(* CODESYS project SingleElevator.project

Project tree, tasks and I/O mapping:
  Device : CODESYS Control Win V3, 3S - Smart Software Solutions GmbH, version 3.5.18.0
    application Application
      libraries: Standard, 3.5.18.0 (System)
      task MainTask (cyclic, interval t#20ms, priority 1) calls Simulation, GA_collector, PLC_PRG
      task VISU_TASK (cyclic, interval 100 ms, priority 31) calls VisuElems.Visu_Prg
      global variables GVL
      visualisation Visualization
      program Simulation [ST]
      function block Doors_GA [SFC]: _aReady_active, _aBusy_active, _aChiusura_active, _aApertura_active, _aApertura_exit, _aOpFinished_active, _aResetDone_active, _aChiusura_exit_1, _a_aInit_activeState
      program GA_collector [FBD]
      function block MovimentoVert_GA [SFC]: _aInit_active, _aReady_active, _aBusy_active, _aSalita_active, _aDiscesa_active, _aSalita_exit, _aDiscesa_exit
      program PLC_PRG [SFC]: _aOpenDoors1_active, _aInizio_homing_active, _aFinecorsa_active, _aRisalitaLenta_active, _aOpenDoors_active, _aHMI_wait_active, _aMoto_verticale_exit, _aOpenDoors_exit, _aOpenDoors1_exit, _aMemoria_chiamate_active, _aMoto_verticale_active_1, _aChiusura_P_exit, _aChiusura_P_active, _aMoto_verticale_entry
  text list GlobalTextList
*)

// Device/Application/GVL
//{attribute 'qualified_only'}
VAR_GLOBAL
(* Elevator managing variables*)
	Open: BOOL;				(* Sensor: the door is fully open*)
	Closed: BOOL;			(* Sensor: the door is fully closed*)
	LimitDown: BOOL;		(* Sensor: lower limit sensor, if TRUE the lift has reached the lower limit*)
	LimitUp: BOOL;			(* Sensor: upper limit sensor, if TRUE the lift has reached the upper limit*)
	DeckSensor: BOOL;		(* Sensor: if TRUE the cab is in proximity of a deck*)
	RampSensor: BOOL;		(* Sensor: if TRUE the cab is in proximity of a ramp*)
	Presence :BOOL; 		(* Sensor: if TRUE something blocks the door photocell*)
	Emergency: BOOL;		(* Input: if TRUE the emergency button has been pressed*)

	Closing: BOOL;			(* Actuator: if TRUE the door starts closing*)
	Opening: BOOL;			(* Actuator: the door starts opening*)
	Motor_on: BOOL;			(* Actuator: if TRUE the lift pulley motor start moving*)
	Up: BOOL;				(* Actuator parameter: if TRUE the lift moves upward, downward otherwise*)
	Vel: BOOL;				(* Actuator parameter: motor speed, if TRUE high speed, low speed otherwise*)


	Current: INT;  			(* Visualization: variable used to storage the current deck*)
    Destination: INT;		(* Visualization: variable used to storage the the destination deck*)
	EmergencyVis: BOOL; 	(* Visualization: if TRUE the emergency light is turned on*)

	InitialDeck: INT := 1;	(* Only for simulation: variable used to define the initial deck*)
	InitCycle: BOOL := FALSE;(* Only for simulation: used to execute the instruction at the first cycle*)
	Height: INT;			(* Only for simulation: elevator height*)
	DeckRest: INT;        	(* Only for simulation: division rest for generating deck sensor*)
	Memory: INT;
	RampRest: INT;			(* Only for simulation: division rest for generating the ramp position*)
	MemoryR: INT;
	Door: INT;				(* Only for simulation: to visualize the closing of the door*)
	Displacement: INT;		(* Only for simulation: lift displacement, dependent on the motor speed*)

 (*Inputs: internal panel variables*)
	PG: BOOL;
	P1: BOOL;
	P2: BOOL;
	P3: BOOL;
	P4: BOOL;
	P5: BOOL;
	P6: BOOL;
	P7: BOOL;

(*Visualization: internal panel variables used to turn on the LED*)
	PGVis: BOOL;
	P1Vis: BOOL;
	P2Vis: BOOL;
	P3Vis: BOOL;
	P4Vis: BOOL;
	P5Vis: BOOL;
	P6Vis: BOOL;
	P7Vis: BOOL;

(*Inputs: external panel variables*)
	UpDeckG: BOOL;
	UpDeck1: BOOL;
	UpDeck2: BOOL;
	UpDeck3: BOOL;
	UpDeck4: BOOL;
	UpDeck5: BOOL;
	UpDeck6: BOOL;
	DownDeck7: BOOL;
	DownDeck6: BOOL;
	DownDeck5: BOOL;
	DownDeck4: BOOL;
	DownDeck3: BOOL;
	DownDeck2: BOOL;
	DownDeck1: BOOL;

(*Visualization: external panel variables used to turn on the LED*)
	UpDeckGVis: BOOL;
	UpDeck1Vis: BOOL;
	UpDeck2Vis: BOOL;
	UpDeck3Vis: BOOL;
	UpDeck4Vis: BOOL;
	UpDeck5Vis: BOOL;
	UpDeck6Vis: BOOL;
	DownDeck7Vis: BOOL;
	DownDeck6Vis: BOOL;
	DownDeck5Vis: BOOL;
	DownDeck4Vis: BOOL;
	DownDeck3Vis: BOOL;
	DownDeck2Vis: BOOL;
	DownDeck1Vis: BOOL;

(*Only for simulation: variables used to simulate the fault on deck sensor*)
	SensorG: BOOL;				(* if TRUE the magnetic information for deck G is lost and the deck sensor cannot become TRUE*)
	Sensor1: BOOL;				(* if TRUE the magnetic information for deck 1 is lost and the deck sensor cannot become TRUE*)
	Sensor2: BOOL;
	Sensor3: BOOL;
	Sensor4: BOOL;
	Sensor5: BOOL;
	Sensor6: BOOL;
	Sensor7: BOOL;
	FaultSensorAlarm: BOOL; 	(* Visulaization: if TRUE alerts the user of a deck sensor fault*)

(*Only for simulation: variables used to simulate the fault on ramp sensor*)
	RampGUp: BOOL;
	Ramp1Down: BOOL;
	Ramp1Up:BOOL;
	Ramp2Down: BOOL;
	Ramp2Up:BOOL;
	Ramp3Down: BOOL;
	Ramp3Up:BOOL;
	Ramp4Down: BOOL;
	Ramp4Up:BOOL;
	Ramp5Down: BOOL;
	Ramp5Up:BOOL;
	Ramp6Down: BOOL;
	Ramp6Up:BOOL;
	Ramp7Down: BOOL;
	FaultRampAlarm: BOOL; 		(* Visulaization: if TRUE alerts the user of a ramp sensor fault*)
	SensorGOK: BOOL;
	Sensor1OK: BOOL;
	Sensor2OK: BOOL;
	Sensor6OK: BOOL;
	Sensor3OK: BOOL;
	Sensor4OK: BOOL;
	Sensor5OK: BOOL;
	Sensor7OK: BOOL;
	RampGUpOK: BOOL;
	Ramp1DownOK: BOOL;
	Ramp1UpOK: BOOL;
	Ramp2DownOK: BOOL;
	Ramp2UpOK: BOOL;
	Ramp3DownOK: BOOL;
	Ramp3UpOK: BOOL;
	Ramp4DownOK: BOOL;
	Ramp4UpOK: BOOL;
	Ramp5DownOK: BOOL;
	Ramp5UpOK: BOOL;
	Ramp6DownOK: BOOL;
	Ramp6UpOK: BOOL;
	Ramp7DownOK: BOOL;
	Ramp7UpOK: BOOL;
	Doors_GA_0: Doors_GA;
	MovimentoVert_GA_0: MovimentoVert_GA;
	Homing: BOOL;
END_VAR

// Device/Application/Simulation
PROGRAM Simulation
VAR
END_VAR

(* Initial position of the cab inside the hoistway. It is executed only at the first cycle.  *)
IF NOT GVL.InitCycle THEN
			GVL.InitCycle := TRUE ;
			GVL.Height := 20 * GVL.InitialDeck;
		    GVL.Door := 0;
			GVL.Current := GVL.Height / 20;
END_IF;

(* Elevator management, these instructions are executed each cycle time*)

(* Elevator door control. *)
IF GVL.Closing THEN
	GVL.Door := GVL.Door + 1;		(*Closing door management*)
	GVL.Open := FALSE;
END_IF

IF GVL.Door >= 60 THEN						(* Closed door limit*)
	GVL.Closed := TRUE;
END_IF

IF GVL.Opening THEN
	GVL.Door := GVL.Door - 1; 	(* Opening door management*)
	GVL.Closed := FALSE;
END_IF

IF GVL.Door <= 0 THEN							(* Open door limit*)
	GVL.Open := TRUE;
END_IF


(* Maximum and minimum management in the door simulation*)
IF GVL.Door < 0 THEN
	 GVL.Door := 0;
END_IF

IF GVL.Door > 60 THEN
	GVL.Door := 60;
END_IF


(* Control of the cab position inside the hostway. *)
(* Displacement definition for graphic visualization*)
IF GVL.Vel THEN 
	GVL.Displacement := 2;
ELSE 
	GVL.Displacement := 1;
END_IF


(* Height modification relying on direction and speed*)
IF GVL.Motor_on AND GVL.Up THEN
	GVL.Height := GVL.Height + GVL.Displacement;
	GVL.LimitDown := FALSE;
END_IF

IF GVL.Motor_on AND NOT GVL.Up THEN
	GVL.Height := GVL.Height - GVL.Displacement;
	GVL.LimitUp := FALSE;
END_IF


(* Limits for visualization*)
IF GVL.Height < -20 THEN
	GVL.Height := -20;
END_IF

IF GVL.Height > 160 THEN
	GVL.Height := 160;
END_IF

(* Limit sensors management*)
IF GVL.Height <= -10 THEN
	GVL.LimitDown := TRUE;
END_IF

IF GVL.Height >= 150 THEN
	 GVL.LimitUp := TRUE;
END_IF


(*-------------------------------------------------------------------*)
(*  Fault Management (Deck and Ramp Sensors)   *)
(*-------------------------------------------------------------------*)
(* Deck Sensor*)
(* Range of value where the deck sensor is active*)
IF ((GVL.Height >= -1) AND (GVL.Height <= 1)) THEN
	GVL.SensorGOK := TRUE;
ELSE  
	GVL.SensorGOK := FALSE;
END_IF

IF ((GVL.Height >= 20-1) AND (GVL.Height <= 20+1)) THEN
	GVL.Sensor1OK := TRUE;
ELSE  
	GVL.Sensor1OK := FALSE;
END_IF

IF ((GVL.Height >= 40-1) AND (GVL.Height <= 40+1)) THEN
	GVL.Sensor2OK := TRUE;
ELSE  
	GVL.Sensor2OK := FALSE;
END_IF

IF ((GVL.Height >= 60-1) AND (GVL.Height <= 60+1)) THEN
	GVL.Sensor3OK := TRUE;
ELSE  
	GVL.Sensor3OK := FALSE;
END_IF

IF ((GVL.Height >= 80-1) AND (GVL.Height <= 80+1)) THEN
	GVL.Sensor4OK := TRUE;
ELSE  
	GVL.Sensor4OK := FALSE;
END_IF

IF ((GVL.Height >= 100-1) AND (GVL.Height <= 100+1)) THEN
	GVL.Sensor5OK := TRUE;
ELSE   
	GVL.Sensor5OK := FALSE;
END_IF

IF ((GVL.Height >= 120-1) AND (GVL.Height <= 120+1)) THEN
	GVL.Sensor6OK := TRUE;
ELSE  
	GVL.Sensor6OK := FALSE;
END_IF

IF ((GVL.Height >= 140-1) AND (GVL.Height <= 140+1)) THEN
	GVL.Sensor7OK := TRUE;
ELSE  
	GVL.Sensor7OK := FALSE;
END_IF

GVL.DeckSensor := (GVL.SensorGOK AND NOT GVL.SensorG) OR
				    (GVL.Sensor1OK AND NOT GVL.Sensor1) OR
				    (GVL.Sensor2OK AND NOT GVL.Sensor2) OR
				    (GVL.Sensor3OK AND NOT GVL.Sensor3) OR
				    (GVL.Sensor4OK AND NOT GVL.Sensor4) OR
				    (GVL.Sensor5OK AND NOT GVL.Sensor5) OR
				    (GVL.Sensor6OK AND NOT GVL.Sensor6) OR
				    (GVL.Sensor7OK AND NOT GVL.Sensor7);

(* Ramp Sensor*)
(* Range of value where the ramp sensor is active*)
IF ((GVL.Height >= 5-1) AND (GVL.Height <= 5+1)) THEN
	GVL.RampGUpOK := TRUE;
ELSE 
	GVL.RampGUpOK := FALSE;
END_IF

(* Ramp close to deck 1*)
IF ((GVL.Height >= 15-1) AND (GVL.Height <= 15+1)) THEN
	GVL.Ramp1DownOK := TRUE;
ELSE 
	GVL.Ramp1DownOK := FALSE;
END_IF

IF ((GVL.Height >= 25-1) AND (GVL.Height <= 25+1)) THEN
	GVL.Ramp1UpOK := TRUE;
ELSE 
	GVL.Ramp1UpOK := FALSE;
END_IF

(* Ramp close to deck 2*)
IF ((GVL.Height >= 35-1) AND (GVL.Height <= 35+1)) THEN
	GVL.Ramp2DownOK := TRUE;
ELSE 
	GVL.Ramp2DownOK := FALSE;
END_IF

IF ((GVL.Height >= 45-1) AND (GVL.Height <= 45+1)) THEN
	GVL.Ramp2UpOK := TRUE;
ELSE 
	GVL.Ramp2UpOK := FALSE;
END_IF

(*Ramp close to deck  3*)
IF ((GVL.Height >= 55-1) AND (GVL.Height <= 55+1)) THEN
	GVL.Ramp3DownOK := TRUE;
ELSE 
	GVL.Ramp3DownOK := FALSE;
END_IF

IF ((GVL.Height >= 65-1) AND (GVL.Height <= 65+1)) THEN
	GVL.Ramp3UpOK := TRUE;
ELSE 
	GVL.Ramp3UpOK := FALSE;
END_IF

(* Ramp close to deck  4*)
IF ((GVL.Height >= 75-1) AND (GVL.Height <= 75+1)) THEN
	GVL.Ramp4DownOK := TRUE;
ELSE 
	GVL.Ramp4DownOK := FALSE;
END_IF

IF ((GVL.Height >= 85-1) AND (GVL.Height <= 85+1)) THEN
	GVL.Ramp4UpOK := TRUE;
ELSE 
	GVL.Ramp4UpOK:=FALSE;
END_IF

(* Ramp close to deck  5*)
IF ((GVL.Height >= 95-1) AND (GVL.Height <= 95+1)) THEN
	GVL.Ramp5DownOK := TRUE;
ELSE 
	GVL.Ramp5DownOK := FALSE;
END_IF

IF ((GVL.Height >= 105-1) AND (GVL.Height <= 105+1)) THEN
	GVL.Ramp5UpOK := TRUE;
ELSE
	GVL.Ramp5UpOK := FALSE;
END_IF

(* Ramp close to deck  6*)
IF ((GVL.Height >= 115-1) AND (GVL.Height <= 115+1)) THEN
	GVL.Ramp6DownOK := TRUE;
ELSE 
	GVL.Ramp6DownOK := FALSE;
END_IF

IF ((GVL.Height >= 125-1) AND (GVL.Height <= 125+1)) THEN
	GVL.Ramp6UpOK := TRUE;
ELSE 
	GVL.Ramp6UpOK := FALSE;
END_IF

(* Ramp close to deck  7*)
IF ((GVL.Height >= 135-1) AND (GVL.Height <= 135+1)) THEN
	GVL.Ramp7DownOK := TRUE;
ELSE 
	GVL.Ramp7DownOK := FALSE;
END_IF

GVL.RampSensor:=(GVL.RampGUpOK AND NOT GVL.RampGUp) OR 
								(GVL.Ramp1DownOK AND NOT GVL.Ramp1Down ) OR 
								(GVL.Ramp1UpOK AND NOT GVL.Ramp1Up ) OR
								(GVL.Ramp2DownOK AND NOT GVL.Ramp2Down ) OR 
								(GVL.Ramp2UpOK AND NOT GVL.Ramp2Up ) OR
								(GVL.Ramp3DownOK AND NOT GVL.Ramp3Down ) OR
 								(GVL.Ramp3UpOK AND NOT GVL.Ramp3Up ) OR
								(GVL.Ramp4DownOK AND NOT GVL.Ramp4Down ) OR
 								(GVL.Ramp4UpOK AND NOT GVL.Ramp4Up ) OR
								(GVL.Ramp5DownOK AND NOT GVL.Ramp5Down ) OR
 								(GVL.Ramp5UpOK AND NOT GVL.Ramp5Up ) OR
								(GVL.Ramp6DownOK AND NOT GVL.Ramp6Down ) OR
								(GVL.Ramp6UpOK AND NOT GVL.Ramp6Up ) OR
								(GVL.Ramp7DownOK AND NOT GVL.Ramp7Down );

END_PROGRAM

// Device/Application/GA_collector
PROGRAM GA_collector
VAR
END_VAR

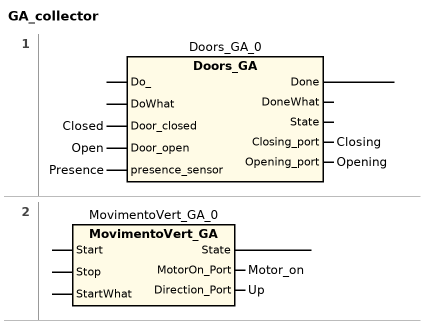
// NETWORK 1
Doors_GA_0(
    Door_closed := Closed,
    Door_open := Open,
    presence_sensor := Presence,
    Closing_port => Closing,
    Opening_port => Opening); // Doors_GA

// NETWORK 2
MovimentoVert_GA_0(MotorOn_Port => Motor_on, Direction_Port => Up); // MovimentoVert_GA

END_PROGRAM

// Device/Application/Doors_GA
FUNCTION_BLOCK Doors_GA
VAR_INPUT
	Do_: BOOL;
	DoWhat: STRING;
	Door_closed: BOOL;
	Door_open: BOOL;
	presence_sensor: BOOL;
END_VAR
VAR_OUTPUT
	Done: BOOL;
	DoneWhat: STRING;
    State: STRING;
	Closing_port: BOOL;
	Opening_port: BOOL;
END_VAR
VAR
END_VAR

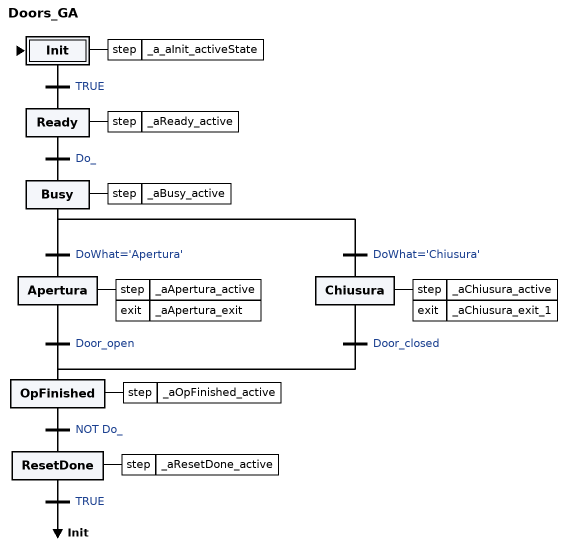
INITIAL_STEP Init:
    _a_aInit_activeState(N);  // step action
END_STEP
TRANSITION FROM Init TO Ready
    := TRUE;
END_TRANSITION
STEP Ready:
    _aReady_active(N);  // step action
END_STEP
TRANSITION FROM Ready TO Busy
    := Do_;
END_TRANSITION
STEP Busy:
    _aBusy_active(N);  // step action
END_STEP
TRANSITION FROM Busy TO Apertura
    := DoWhat='Apertura';
END_TRANSITION
STEP Apertura:
    _aApertura_active(N);  // step action
    _aApertura_exit(P0);  // exit action
END_STEP
TRANSITION FROM Apertura TO OpFinished
    := Door_open;
END_TRANSITION
TRANSITION FROM Busy TO Chiusura
    := DoWhat='Chiusura';
END_TRANSITION
STEP Chiusura:
    _aChiusura_active(N);  // step action
    _aChiusura_exit_1(P0);  // exit action
END_STEP
TRANSITION FROM Chiusura TO OpFinished
    := Door_closed;
END_TRANSITION
STEP OpFinished:
    _aOpFinished_active(N);  // step action
END_STEP
TRANSITION FROM OpFinished TO ResetDone
    := NOT Do_;
END_TRANSITION
STEP ResetDone:
    _aResetDone_active(N);  // step action
END_STEP
TRANSITION FROM ResetDone TO Init
    := TRUE;
END_TRANSITION

ACTION _aReady_active:
State := 'ready';
END_ACTION

ACTION _aBusy_active:
State := 'Busy';
END_ACTION

ACTION _aChiusura_active:
IF presence_sensor=FALSE AND Door_open=TRUE THEN
Closing_port:=TRUE;
Opening_port:=FALSE;
END_IF

IF presence_sensor= FALSE AND Door_closed=TRUE THEN
Closing_port:=FALSE;
END_IF

IF presence_sensor=TRUE THEN
	Closing_port:=FALSE;
	IF Door_open=FALSE THEN
    Opening_port:=TRUE;
	END_IF
	IF Door_open=TRUE THEN
	Opening_port:=FALSE;
	END_IF
END_IF
END_ACTION

ACTION _aApertura_active:
Opening_port :=TRUE;
END_ACTION

ACTION _aApertura_exit:
Opening_port := FALSE;
END_ACTION

ACTION _aOpFinished_active:
Done := TRUE;

IF door_open=TRUE THEN
	DoneWhat:='apertura';
END_IF

IF door_closed=TRUE THEN
	DoneWhat:='chiusura';
END_IF
END_ACTION

ACTION _aResetDone_active:
Done:=FALSE;
END_ACTION

ACTION _aChiusura_exit_1:
Closing_port := FALSE;
END_ACTION

ACTION _a_aInit_activeState:
State :='init';
END_ACTION

END_FUNCTION_BLOCK

// Device/Application/MovimentoVert_GA
FUNCTION_BLOCK MovimentoVert_GA
VAR_INPUT
	Start: BOOL;
	Stop: BOOL;
	StartWhat: STRING;
END_VAR
VAR_OUTPUT
	State: STRING;
	MotorOn_Port: BOOL;
	Direction_Port: BOOL;
END_VAR
VAR
END_VAR

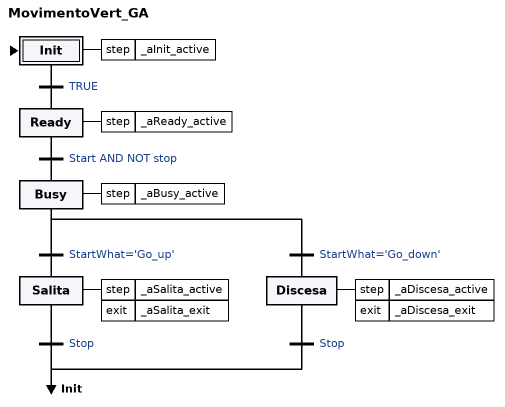
INITIAL_STEP Init:
    _aInit_active(N);  // step action
END_STEP
TRANSITION FROM Init TO Ready
    := TRUE;
END_TRANSITION
STEP Ready:
    _aReady_active(N);  // step action
END_STEP
TRANSITION FROM Ready TO Busy
    := Start AND NOT stop;
END_TRANSITION
STEP Busy:
    _aBusy_active(N);  // step action
END_STEP
TRANSITION FROM Busy TO Salita
    := StartWhat='Go_up';
END_TRANSITION
STEP Salita:
    _aSalita_active(N);  // step action
    _aSalita_exit(P0);  // exit action
END_STEP
TRANSITION FROM Salita TO Init
    := Stop;
END_TRANSITION
TRANSITION FROM Busy TO Discesa
    := StartWhat='Go_down';
END_TRANSITION
STEP Discesa:
    _aDiscesa_active(N);  // step action
    _aDiscesa_exit(P0);  // exit action
END_STEP
TRANSITION FROM Discesa TO Init
    := Stop;
END_TRANSITION

ACTION _aInit_active:
State:='init';
END_ACTION

ACTION _aReady_active:
State:='Ready';
END_ACTION

ACTION _aBusy_active:
State:='Busy';
END_ACTION

ACTION _aSalita_active:
Direction_Port := TRUE;
MotorOn_Port := TRUE;
END_ACTION

ACTION _aDiscesa_active:
Direction_Port := FALSE;
MotorOn_Port := TRUE;
END_ACTION

ACTION _aSalita_exit:
MotorOn_Port := FALSE;
END_ACTION

ACTION _aDiscesa_exit:
MotorOn_Port := FALSE;
END_ACTION

END_FUNCTION_BLOCK

// Device/Application/PLC_PRG
PROGRAM PLC_PRG
VAR
	OpComplete: BOOL;
	OpFinished: BOOL;
	OpDone: BOOL;
	OperationComplete: BOOL;
	Richiesta: BOOL;
	Coerent: INT;
	Libera: BOOL;
	OpFatta: BOOL;
	Current_Ok: BOOL;
	t_deck: INT := 0;
	Apertura_completata: BOOL;
	RR: INT;
	Check1: BOOL;
	RS_counter: INT := 0;
	Piano_partenza: INT;
	ok: BOOL;
	t_ramp: INT := 0;
	NuovaRichiesta: INT;
	Chiamata_in_sospeso: BOOL;
	VecchiaRichiesta: INT;
	Request_up: BOOL;
	Request_down: BOOL;
	Richiesta_interna: BOOL;
	RichiestaG: INT;
	Richiesta1: INT;
	Richiesta2: INT;
	Richiesta3: INT;
	Richiesta4: INT;
	Deck_counter: INT := 0;
	Ramp_counter: INT := 0;
	D_counter: INT := 0;
	t_finecorsa_alto: INT := 0;
	t_finecorsa_basso: INT := 0;
END_VAR

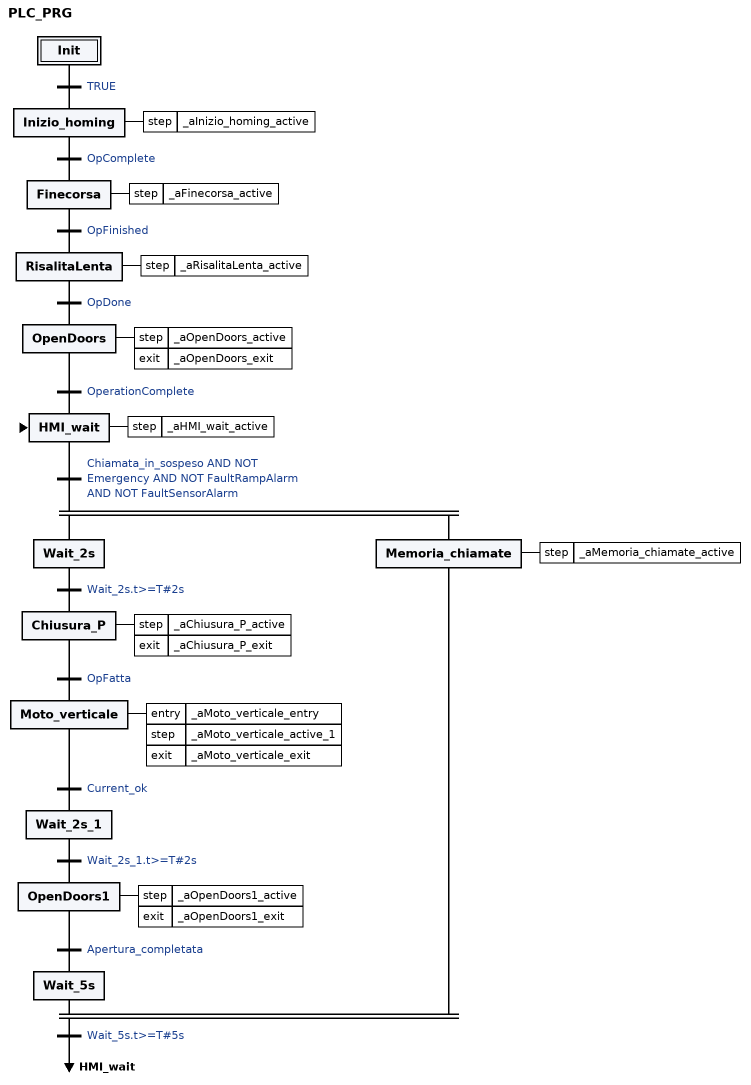
INITIAL_STEP Init:
END_STEP
TRANSITION FROM Init TO Inizio_homing
    := TRUE;
END_TRANSITION
STEP Inizio_homing:
    _aInizio_homing_active(N);  // step action
END_STEP
TRANSITION FROM Inizio_homing TO Finecorsa
    := OpComplete;
END_TRANSITION
STEP Finecorsa:
    _aFinecorsa_active(N);  // step action
END_STEP
TRANSITION FROM Finecorsa TO RisalitaLenta
    := OpFinished;
END_TRANSITION
STEP RisalitaLenta:
    _aRisalitaLenta_active(N);  // step action
END_STEP
TRANSITION FROM RisalitaLenta TO OpenDoors
    := OpDone;
END_TRANSITION
STEP OpenDoors:
    _aOpenDoors_active(N);  // step action
    _aOpenDoors_exit(P0);  // exit action
END_STEP
TRANSITION FROM OpenDoors TO HMI_wait
    := OperationComplete;
END_TRANSITION
STEP HMI_wait:
    _aHMI_wait_active(N);  // step action
END_STEP
TRANSITION FROM HMI_wait TO (Wait_2s, Memoria_chiamate)
    := Chiamata_in_sospeso AND NOT Emergency AND NOT FaultRampAlarm AND NOT FaultSensorAlarm;
END_TRANSITION
STEP Wait_2s:
END_STEP
TRANSITION FROM Wait_2s TO Chiusura_P
    := Wait_2s.t>=T#2s;
END_TRANSITION
STEP Chiusura_P:
    _aChiusura_P_active(N);  // step action
    _aChiusura_P_exit(P0);  // exit action
END_STEP
TRANSITION FROM Chiusura_P TO Moto_verticale
    := OpFatta;
END_TRANSITION
STEP Moto_verticale:
    _aMoto_verticale_entry(P1);  // entry action
    _aMoto_verticale_active_1(N);  // step action
    _aMoto_verticale_exit(P0);  // exit action
END_STEP
TRANSITION FROM Moto_verticale TO Wait_2s_1
    := Current_ok;
END_TRANSITION
STEP Wait_2s_1:
END_STEP
TRANSITION FROM Wait_2s_1 TO OpenDoors1
    := Wait_2s_1.t>=T#2s;
END_TRANSITION
STEP OpenDoors1:
    _aOpenDoors1_active(N);  // step action
    _aOpenDoors1_exit(P0);  // exit action
END_STEP
TRANSITION FROM OpenDoors1 TO Wait_5s
    := Apertura_completata;
END_TRANSITION
STEP Wait_5s:
END_STEP
STEP Memoria_chiamate:
    _aMemoria_chiamate_active(N);  // step action
END_STEP
TRANSITION FROM (Wait_5s, Memoria_chiamate) TO HMI_wait
    := Wait_5s.t>=T#5s;
END_TRANSITION

ACTION _aOpenDoors1_active:
IF Doors_GA_0.State='ready' THEN
	Doors_GA_0.Do_:=TRUE;
	Doors_GA_0.DoWhat:='Apertura';
END_IF

IF (Doors_GA_0.Done= TRUE) AND Doors_GA_0.State='Busy' THEN
	Doors_GA_0.Do_:=FALSE;
	Apertura_completata:=TRUE;
END_IF
END_ACTION

ACTION _aInizio_homing_active:
IF Doors_GA_0.State='ready' THEN
	Doors_GA_0.Do_:=TRUE;
	Doors_GA_0.DoWhat:='Chiusura';
END_IF

IF Doors_GA_0.Done= TRUE AND Doors_GA_0.State='Busy' THEN
	Doors_GA_0.Do_:=FALSE;
	OpComplete:=TRUE;
END_IF
END_ACTION

ACTION _aFinecorsa_active:
IF (LimitDown= FALSE) AND MovimentoVert_GA_0.State='Ready' THEN
    Vel:=FALSE;
	MovimentoVert_GA_0.Start:= TRUE;
	MovimentoVert_GA_0.StartWhat:='Go_down';
END_IF

IF LimitDown= TRUE THEN
	MovimentoVert_GA_0.Stop:= TRUE;
	OpFinished:= TRUE;
END_IF
END_ACTION

ACTION _aRisalitaLenta_active:
Vel:=FALSE;
IF MovimentoVert_GA_0.State='Ready'THEN
 IF DeckSensor= FALSE THEN
	MovimentoVert_GA_0.Stop:=FALSE;
	MovimentoVert_GA_0.Start:=TRUE;
	MovimentoVert_GA_0.StartWhat:='Go_up';
 END_IF
END_IF

IF DeckSensor= TRUE THEN
	MovimentoVert_GA_0.Stop:= TRUE;
	OpDone:=TRUE;
END_IF

//INIZIALIZZAZIONE
Current:=-1;
Chiamata_in_sospeso:=FALSE;
Current_Ok:=FALSE;
Richiesta:=FALSE;
END_ACTION

ACTION _aOpenDoors_active:
IF Doors_GA_0.State='ready' THEN
	Doors_GA_0.Do_:=TRUE;
	Doors_GA_0.DoWhat:='Apertura';
END_IF

IF (Doors_GA_0.Done= TRUE) AND Doors_GA_0.State='Busy' THEN
	Doors_GA_0.Do_:=FALSE;
	OperationComplete:=TRUE;
END_IF
END_ACTION

ACTION _aHMI_wait_active:
//EMERGENCY
IF Emergency =TRUE THEN
	EmergencyVis:=TRUE;
END_IF
IF Emergency = FALSE THEN
	EmergencyVis:=FALSE;
END_IF


//PULSANTIERA INTERNA

IF Chiamata_in_sospeso= FALSE THEN
	
IF PG= TRUE THEN
    Destination:=0; 
	PGVis:= TRUE;	
	Chiamata_in_sospeso:=TRUE;
END_IF

IF P1= TRUE THEN
    Destination:=1; 
	P1Vis:= TRUE;	
	Chiamata_in_sospeso:=TRUE;
END_IF

IF P2= TRUE THEN
    Destination:=2; 
	P2Vis:= TRUE;
	Chiamata_in_sospeso:=TRUE;
END_IF

IF P3= TRUE THEN
    Destination:=3; 
	P3Vis:= TRUE;	
	Chiamata_in_sospeso:=TRUE;
END_IF

IF P4= TRUE THEN
    Destination:=4; 
	P4Vis:= TRUE;	
	Chiamata_in_sospeso:=TRUE;
END_IF

IF P5= TRUE THEN
    Destination:=5; 
	P5Vis:= TRUE;	
	Chiamata_in_sospeso:=TRUE;
END_IF

IF P6= TRUE THEN
    Destination:=6; 
	P6Vis:= TRUE;	
	Chiamata_in_sospeso:=TRUE;
END_IF

IF P7=TRUE THEN
    Destination:=7; 
	P7Vis:= TRUE;	
	Chiamata_in_sospeso:=TRUE;
END_IF
END_IF
//Pulsantiera interna end

//Pulsantiera esterna, inizio up

IF UpDeckG=TRUE THEN
	UpDeckGVis:=TRUE;
    IF Chiamata_in_sospeso=FALSE THEN
	Destination:=0;
	Chiamata_in_sospeso:=TRUE;
	END_IF
END_IF

IF UpDeck1=TRUE THEN
	UpDeck1Vis:=TRUE;
    IF Chiamata_in_sospeso=FALSE THEN
	Destination:=1;
	Chiamata_in_sospeso:=TRUE;
	END_IF
END_IF

IF UpDeck2=TRUE THEN
	UpDeck2Vis:=TRUE;
    IF Chiamata_in_sospeso=FALSE THEN
	Destination:=2;
	Chiamata_in_sospeso:=TRUE;
	END_IF
END_IF

IF UpDeck3=TRUE THEN
	UpDeck3Vis:=TRUE;
    IF Chiamata_in_sospeso=FALSE THEN
	Destination:=3;
	Chiamata_in_sospeso:=TRUE;
	END_IF
END_IF

IF UpDeck4=TRUE THEN
	UpDeck4Vis:=TRUE;
    IF Chiamata_in_sospeso=FALSE THEN
	Destination:=4;
	Chiamata_in_sospeso:=TRUE;
	END_IF
END_IF

IF UpDeck5=TRUE THEN
	UpDeck5Vis:=TRUE;
    IF Chiamata_in_sospeso=FALSE THEN
	Destination:=5;
	Chiamata_in_sospeso:=TRUE;
	END_IF
END_IF

IF UpDeck6=TRUE THEN
	UpDeck6Vis:=TRUE;
    IF Chiamata_in_sospeso=FALSE THEN
	Destination:=6;
	Chiamata_in_sospeso:=TRUE;
	END_IF
END_IF

//Inizio down

IF DownDeck1=TRUE THEN
	DownDeck1Vis:=TRUE;
    IF Chiamata_in_sospeso=FALSE THEN
	Destination:=1;
	Chiamata_in_sospeso:=TRUE;
	END_IF
END_IF

IF DownDeck2=TRUE THEN
	DownDeck2Vis:=TRUE;
    IF Chiamata_in_sospeso=FALSE THEN
	Destination:=2;
	Chiamata_in_sospeso:=TRUE;
	END_IF
END_IF

IF DownDeck3=TRUE THEN
	DownDeck3Vis:=TRUE;
    IF Chiamata_in_sospeso=FALSE THEN
	Destination:=3;
	Chiamata_in_sospeso:=TRUE;
	END_IF
END_IF

IF DownDeck4=TRUE THEN
	DownDeck4Vis:=TRUE;
    IF Chiamata_in_sospeso=FALSE THEN
	Destination:=4;
	Chiamata_in_sospeso:=TRUE;
	END_IF
END_IF

IF DownDeck5=TRUE THEN
	DownDeck5Vis:=TRUE;
    IF Chiamata_in_sospeso=FALSE THEN
	Destination:=5;
	Chiamata_in_sospeso:=TRUE;
	END_IF
END_IF

IF DownDeck6=TRUE THEN
	DownDeck6Vis:=TRUE;
    IF Chiamata_in_sospeso=FALSE THEN
	Destination:=6;
	Chiamata_in_sospeso:=TRUE;
	END_IF
END_IF

IF DownDeck7=TRUE THEN
	DownDeck7Vis:=TRUE;
    IF Chiamata_in_sospeso=FALSE THEN
	Destination:=7;
	Chiamata_in_sospeso:=TRUE;
	END_IF
END_IF

//CHIAMATE IN SOSPESO TRAMITE VISUALIZER
IF  PGVis = TRUE
    OR	P1Vis = TRUE 
    OR	P2Vis = TRUE 
    OR	P3Vis = TRUE 
    OR  P4Vis = TRUE 
    OR  P5Vis = TRUE 
    OR	P6Vis = TRUE 
    OR	P7Vis = TRUE
	OR UpDeckGVis = TRUE
	OR UpDeck1Vis = TRUE
	OR UpDeck2Vis = TRUE
	OR UpDeck3Vis = TRUE
	OR UpDeck4Vis = TRUE
	OR UpDeck5Vis = TRUE
	OR UpDeck6Vis = TRUE
	OR DownDeck7Vis = TRUE
	OR DownDeck6Vis = TRUE
	OR DownDeck5Vis = TRUE
	OR DownDeck4Vis = TRUE
	OR DownDeck3Vis = TRUE
	OR DownDeck2Vis = TRUE
	OR DownDeck1Vis = TRUE THEN
	Chiamata_in_sospeso:=TRUE;
	ELSIF PGVis = FALSE
    OR	P1Vis = FALSE 
    OR	P2Vis = FALSE 
    OR	P3Vis = FALSE 
    OR  P4Vis = FALSE 
    OR  P5Vis = FALSE 
    OR	P6Vis = FALSE 
    OR	P7Vis = FALSE
	OR UpDeckGVis = FALSE
	OR UpDeck1Vis = FALSE
	OR UpDeck2Vis = FALSE
	OR UpDeck3Vis = FALSE
	OR UpDeck4Vis = FALSE
	OR UpDeck5Vis = FALSE
	OR UpDeck6Vis = FALSE
	OR DownDeck7Vis = FALSE
	OR DownDeck6Vis = FALSE
	OR DownDeck5Vis = FALSE
	OR DownDeck4Vis = FALSE
	OR DownDeck3Vis = FALSE
	OR DownDeck2Vis = FALSE
	OR DownDeck1Vis = FALSE THEN
	Chiamata_in_sospeso:=FALSE;
END_IF

(*IF Chiamata_in_sospeso=FALSE AND Current=-1 THEN
	Destination:=Current+1;
	ELSIF Current>-1 THEN Destination:=Current;
END_IF*)
END_ACTION

ACTION _aMoto_verticale_exit:
Richiesta:=FALSE;
END_ACTION

ACTION _aOpenDoors_exit:
OperationComplete:=FALSE;
Current_ok:= FALSE;
END_ACTION

ACTION _aOpenDoors1_exit:
Apertura_completata:=FALSE;
RS_counter:=0;

//Se abbiamo raggiunto il piano dobbiamo disattivare i led
IF P7Vis=TRUE AND Current=7 (*AND MovimentoVert_GA_0.State='Ready'*) THEN P7Vis:=FALSE;
ELSIF P6Vis=TRUE  AND Current=6 (*AND MovimentoVert_GA_0.State='Ready'*) THEN P6Vis:=FALSE;
ELSIF P5Vis=TRUE  AND Current=5 (*AND MovimentoVert_GA_0.State='Ready'*) THEN P5Vis:=FALSE;
ELSIF P4Vis=TRUE  AND Current=4 (*AND MovimentoVert_GA_0.State='Ready'*) THEN P4Vis:=FALSE;
ELSIF P3Vis=TRUE  AND Current=3 (*AND MovimentoVert_GA_0.State='Ready'*) THEN P3Vis:=FALSE;	
ELSIF P2Vis=TRUE  AND Current=2 (*AND MovimentoVert_GA_0.State='Ready'*) THEN P2Vis:=FALSE;
ELSIF P1Vis=TRUE  AND Current=1 (*AND MovimentoVert_GA_0.State='Ready'*) THEN P1Vis:=FALSE;	
ELSIF PGVis=TRUE  AND Current=0 (*AND MovimentoVert_GA_0.State='Ready'*) THEN PGVis:=FALSE;	
END_IF

IF UpDeck6Vis=TRUE AND Current=6 (*AND MovimentoVert_GA_0.State='Ready'*)  THEN UpDeck6Vis:=FALSE;
ELSIF UpDeck5Vis=TRUE  AND Current=5 (*AND MovimentoVert_GA_0.State='Ready'*)  THEN UpDeck5Vis:=FALSE;
ELSIF UpDeck4Vis=TRUE  AND Current=4 (*AND MovimentoVert_GA_0.State='Ready'*)  THEN UpDeck4Vis:=FALSE;
ELSIF UpDeck3Vis=TRUE  AND Current=3 (*AND MovimentoVert_GA_0.State='Ready'*)  THEN UpDeck3Vis:=FALSE;
ELSIF UpDeck2Vis=TRUE  AND Current=2 (*AND MovimentoVert_GA_0.State='Ready'*)  THEN UpDeck2Vis:=FALSE;
ELSIF UpDeck1Vis=TRUE  AND Current=1 (*AND MovimentoVert_GA_0.State='Ready'*)  THEN UpDeck1Vis:=FALSE;	
ELSIF UpDeckGVis=TRUE  AND Current=0 (*AND MovimentoVert_GA_0.State='Ready'*)  THEN UpDeckGVis:=FALSE;	
END_IF

IF DownDeck7Vis=TRUE  AND Current=7 (*AND MovimentoVert_GA_0.State='Ready'*)  THEN DownDeck7Vis:=FALSE;
ELSIF DownDeck6Vis=TRUE  AND Current=6 (*AND MovimentoVert_GA_0.State='Ready'*)  THEN DownDeck6Vis:=FALSE;
ELSIF DownDeck5Vis=TRUE  AND Current=5 (*AND MovimentoVert_GA_0.State='Ready'*)  THEN DownDeck5Vis:=FALSE;
ELSIF DownDeck4Vis=TRUE  AND Current=4 (*AND MovimentoVert_GA_0.State='Ready'*)  THEN DownDeck4Vis:=FALSE;
ELSIF DownDeck3Vis=TRUE  AND Current=3 (*AND MovimentoVert_GA_0.State='Ready'*)  THEN DownDeck3Vis:=FALSE;
ELSIF DownDeck2Vis=TRUE  AND Current=2 (*AND MovimentoVert_GA_0.State='Ready'*)  THEN DownDeck2Vis:=FALSE;
ELSIF DownDeck1Vis=TRUE  AND Current=1 (*AND MovimentoVert_GA_0.State='Ready'*)  THEN DownDeck1Vis:=FALSE;	
END_IF
END_ACTION

ACTION _aMemoria_chiamate_active:
//EMERGENCY AL VOLO
IF Emergency=TRUE THEN
	IF MovimentoVert_GA_0.StartWhat='Go_up' AND MovimentoVert_GA_0.State='Busy' AND RS_counter<2*(current-piano_partenza) THEN
		VEL:=FALSE;
		IF Current+1<Destination THEN
		Destination:=Current+1;
		END_IF
	END_IF
	
	IF MovimentoVert_GA_0.StartWhat='Go_down' AND MovimentoVert_GA_0.State='Busy' THEN
		VEL:=FALSE;
		IF Current-1>Destination THEN
		Destination:=Current-1;
		END_IF
	END_IF
	
END_IF

//FERMATA PER GUASTO DECK
IF DeckSensor=TRUE THEN
	Deck_counter:=0;
	Ramp_counter:=0;
END_IF

IF Ramp_counter=3 AND Deck_Counter=0 THEN
		VEL:=FALSE;
		FaultSensorAlarm:=TRUE;

	IF MovimentoVert_GA_0.StartWhat='Go_up' AND MovimentoVert_GA_0.State='Busy' THEN
		IF Current+1<Destination THEN
		Destination:=Current+1;
		END_IF
	END_IF
	
	IF MovimentoVert_GA_0.StartWhat='Go_down' AND MovimentoVert_GA_0.State='Busy' THEN
		IF Current-1>Destination THEN
		Destination:=Current-1;
		END_IF
	END_IF
	
END_IF


IF LimitUp=TRUE AND t_finecorsa_alto=0 THEN
	MovimentoVert_GA_0.Stop:=TRUE;
END_IF	

IF LimitUp=TRUE THEN t_finecorsa_alto:=t_finecorsa_alto+1; END_IF

IF LimitUp=TRUE AND t_finecorsa_alto=1 THEN
    Current:=8;
	Destination:=6;
	IF Current_ok=TRUE THEN
		FaultSensorAlarm:=TRUE;
	END_IF
END_IF

IF LimitDown=TRUE AND t_finecorsa_basso=0 THEN
	MovimentoVert_GA_0.Stop:=TRUE;
END_IF

IF LimitDown=TRUE THEN t_finecorsa_basso:=t_finecorsa_basso+1; END_IF

IF LimitDown=TRUE AND t_finecorsa_basso=1 THEN
	Current:=-1;
    Destination:=0;
	IF Current_ok=TRUE THEN
		FaultSensorAlarm:=TRUE;
	END_IF
END_IF

//FERMATA PER GUASTO RAMPA MOTO VERSO L'ALTO
IF RS_counter=1 AND Current=Piano_partenza+1 AND Destination<7 THEN
	VEL:=FALSE;
	FaultRampAlarm:=TRUE;
	Destination:=Current+1;
END_IF

IF RS_counter=3 AND Current=Piano_partenza+2 AND Destination<7 THEN
	VEL:=FALSE;
	FaultRampAlarm:=TRUE;
	Destination:=Current+1;
END_IF

IF RS_counter=5 AND Current=Piano_partenza+3 AND Destination<7 THEN
	VEL:=FALSE;
	FaultRampAlarm:=TRUE;
	Destination:=Current+1;
END_IF

IF RS_counter=7 AND Current=Piano_partenza+4 AND Destination<7 THEN
	VEL:=FALSE;
		FaultRampAlarm:=TRUE;
		Destination:=Current+1;
END_IF

IF RS_counter=9 AND Current=Piano_partenza+5 AND Destination<7 THEN
	VEL:=FALSE;
	FaultRampAlarm:=TRUE;
	IF DeckSensor=TRUE THEN	Destination:=Current+1; END_IF
END_IF

IF RS_counter=11 AND Current=Piano_partenza+6 AND Destination<7 THEN
	VEL:=FALSE;
		FaultRampAlarm:=TRUE;
		Destination:=Current+1;
END_IF

IF RS_counter=13 AND Current=Piano_partenza+7 THEN
	VEL:=FALSE;
	FaultRampAlarm:=TRUE;
END_IF

//FERMATA PER GUASTO RAMPA MOTO VERSO IL BASSO

IF RS_counter=1 AND Current=Piano_partenza-1 AND Destination>0 THEN
	VEL:=FALSE;
		FaultRampAlarm:=TRUE;
		Destination:=Current-1;
END_IF

IF RS_counter=3 AND Current=Piano_partenza-2 AND Destination>0 THEN
	VEL:=FALSE;
		FaultRampAlarm:=TRUE;
		Destination:=Current-1;
END_IF

IF RS_counter=5 AND Current=Piano_partenza-3 AND Destination>0 THEN
	VEL:=FALSE;
		FaultRampAlarm:=TRUE;
		Destination:=Current-1;
END_IF

IF RS_counter=7 AND Current=Piano_partenza-4 AND Destination>0 THEN
	VEL:=FALSE;
		FaultRampAlarm:=TRUE;
		Destination:=Current-1;
END_IF

IF RS_counter=9 AND Current=Piano_partenza-5 AND Destination>0 THEN
	VEL:=FALSE;
		FaultRampAlarm:=TRUE;
		Destination:=Current-1;
END_IF

IF RS_counter=11 AND Current=Piano_partenza-6 AND Destination>0 THEN
	VEL:=FALSE;
		FaultRampAlarm:=TRUE;
		Destination:=Current-1;
END_IF

IF RS_counter=13 AND Current=Piano_partenza-7 THEN
	VEL:=FALSE;
		FaultRampAlarm:=TRUE;
END_IF


//INIZIO PIANI AL VOLO
//Pulsantiera interna	
IF PG= TRUE THEN 
	PGVis:= TRUE;	
	Richiesta_interna:=TRUE;
END_IF

IF P1= TRUE THEN
	P1Vis:= TRUE;	
	Richiesta_interna:=TRUE;
END_IF

IF P2= TRUE THEN 
	P2Vis:= TRUE;
    Richiesta_interna:=TRUE;
END_IF

IF P3= TRUE THEN
	P3Vis:= TRUE;
    Richiesta_interna:=TRUE;
END_IF

IF P4= TRUE THEN
	P4Vis:= TRUE;	
	Richiesta_interna:=TRUE;
END_IF

IF P5= TRUE THEN
	P5Vis:= TRUE;	
	Richiesta_interna:=TRUE;
END_IF

IF P6= TRUE THEN 
	P6Vis:= TRUE;	
	Richiesta_interna:=TRUE;
END_IF

IF P7=TRUE THEN
	P7Vis:= TRUE;	
	Richiesta_interna:=TRUE;
END_IF


//Pulsantiera esterna, inizio up

IF UpDeckG=TRUE THEN
	UpDeckGVis:=TRUE;
    Request_up:=TRUE;
END_IF

IF UpDeck1=TRUE THEN
	UpDeck1Vis:=TRUE;
    Request_up:=TRUE;
END_IF

IF UpDeck2=TRUE THEN
	UpDeck2Vis:=TRUE;
    Request_up:=TRUE;
END_IF

IF UpDeck3=TRUE THEN
	UpDeck3Vis:=TRUE;
    Request_up:=TRUE;
END_IF

IF UpDeck4=TRUE THEN
	UpDeck4Vis:=TRUE;
    Request_up:=TRUE;
END_IF

IF UpDeck5=TRUE THEN
	UpDeck5Vis:=TRUE;
    Request_up:=TRUE;
END_IF

IF UpDeck6=TRUE THEN
	UpDeck6Vis:=TRUE;
    Request_up:=TRUE;
END_IF

//Inizio down

IF DownDeck1=TRUE THEN
	DownDeck1Vis:=TRUE;
    Request_down:=TRUE;
END_IF

IF DownDeck2=TRUE THEN
	DownDeck2Vis:=TRUE;
    Request_down:=TRUE;
END_IF

IF DownDeck3=TRUE THEN
	DownDeck3Vis:=TRUE;
    Request_down:=TRUE;
END_IF

IF DownDeck4=TRUE THEN
	DownDeck4Vis:=TRUE;
    Request_down:=TRUE;
END_IF

IF DownDeck5=TRUE THEN
	DownDeck5Vis:=TRUE;
    Request_down:=TRUE;
END_IF

IF DownDeck6=TRUE THEN
	DownDeck6Vis:=TRUE;
    Request_down:=TRUE;
END_IF

IF DownDeck7=TRUE THEN
	DownDeck7Vis:=TRUE;
    Request_down:=TRUE;
END_IF

//DEFINIZIONE REQUEST

IF DownDeck1Vis=FALSE AND DownDeck2Vis=FALSE AND DownDeck3Vis=FALSE AND DownDeck4Vis=FALSE AND DownDeck5Vis=FALSE AND DownDeck6Vis=FALSE AND DownDeck7Vis=FALSE THEN
    Request_Down:=FALSE;
END_IF 

IF UpDeckGVis=FALSE AND UpDeck1Vis=FALSE AND UpDeck2Vis=FALSE AND UpDeck3Vis=FALSE AND UpDeck4Vis=FALSE AND UpDeck5Vis=FALSE AND UpDeck6Vis=FALSE THEN
    Request_up:=FALSE;
END_IF 

IF PGvis=FALSE AND P1vis=FALSE AND P2vis=FALSE AND P3vis=FALSE AND P4vis=FALSE AND P5vis=FALSE AND P6vis=FALSE AND P7vis=FALSE THEN
    Richiesta_interna:=FALSE;
END_IF 


//CHIAMATE AL VOLO


//VIS INTERNI ALTO

IF MovimentoVert_GA_0.StartWhat='Go_up' AND MovimentoVert_GA_0.State='Busy' THEN
	IF Richiesta_interna=TRUE OR Request_up= TRUE THEN
	IF PGVis=TRUE THEN 
    IF 0<Destination AND Current<0 THEN
		Destination:=0;
		ELSIF 0>Destination AND Current_ok=TRUE THEN Destination:=0;
	END_IF
	END_IF
	END_IF
END_IF

IF MovimentoVert_GA_0.StartWhat='Go_up' AND MovimentoVert_GA_0.State='Busy' THEN
	IF Richiesta_interna=TRUE OR Request_up= TRUE THEN
	IF P1Vis=TRUE THEN 
    IF 1<Destination AND Current<1 THEN
		Destination:=1;
		ELSIF 1>Destination AND Current_ok=TRUE THEN Destination:=1;
	END_IF
	END_IF
	END_IF
END_IF

IF MovimentoVert_GA_0.StartWhat='Go_up' AND MovimentoVert_GA_0.State='Busy' THEN
	IF Richiesta_interna=TRUE OR Request_up= TRUE THEN
	IF P2Vis=TRUE THEN 
    IF 2<Destination AND Current<2 THEN
		Destination:=2;
		ELSIF 2>Destination AND Current_ok=TRUE THEN Destination:=2;
	END_IF
	END_IF
	END_IF
END_IF

IF MovimentoVert_GA_0.StartWhat='Go_up' AND MovimentoVert_GA_0.State='Busy' THEN
	IF Richiesta_interna=TRUE OR Request_up= TRUE THEN
	IF P3Vis=TRUE THEN 
    IF 3<Destination AND Current<3 THEN
		Destination:=3;
		ELSIF 3>Destination AND Current_ok=TRUE THEN Destination:=3;
	END_IF
	END_IF
	END_IF
END_IF

IF MovimentoVert_GA_0.StartWhat='Go_up' AND MovimentoVert_GA_0.State='Busy' THEN
	IF Richiesta_interna=TRUE OR Request_up= TRUE THEN
	IF P4Vis=TRUE THEN 
    IF 4<Destination AND Current<4 THEN
		Destination:=4;
		ELSIF 4>Destination AND Current_ok=TRUE THEN Destination:=4;
	END_IF
	END_IF
	END_IF
END_IF

IF MovimentoVert_GA_0.StartWhat='Go_up' AND MovimentoVert_GA_0.State='Busy' THEN
	IF Richiesta_interna=TRUE OR Request_up= TRUE THEN
	IF P5Vis=TRUE THEN 
    IF 5<Destination AND Current<5 THEN
		Destination:=5;
		ELSIF 5>Destination AND Current_ok=TRUE THEN Destination:=5;
	END_IF
	END_IF
	END_IF
END_IF

IF MovimentoVert_GA_0.StartWhat='Go_up' AND MovimentoVert_GA_0.State='Busy' THEN
	IF Richiesta_interna=TRUE OR Request_up= TRUE THEN
	IF P6Vis=TRUE THEN 
    IF 6<Destination AND Current<6 THEN
		Destination:=6;
		ELSIF 6>Destination AND Current_ok=TRUE THEN Destination:=6;
	END_IF
	END_IF
	END_IF
END_IF

IF MovimentoVert_GA_0.StartWhat='Go_up' AND MovimentoVert_GA_0.State='Busy' THEN
	IF Richiesta_interna=TRUE OR Request_up= TRUE THEN
	IF P7Vis=TRUE THEN 
    IF 7<Destination AND Current<7 THEN
		Destination:=7;
		ELSIF 7>Destination AND Current_ok=TRUE THEN Destination:=7;
	END_IF
	END_IF
	END_IF
END_IF


//VIS INTERNI DOWN
IF MovimentoVert_GA_0.StartWhat='Go_down' AND MovimentoVert_GA_0.State='Busy' THEN
	IF Richiesta_interna=TRUE OR Request_down= TRUE THEN
	IF PGVis=TRUE THEN 
    IF 0>Destination AND Current>0 THEN
		Destination:=0;
		ELSIF 0<Destination AND Current_ok=TRUE THEN Destination:=0;
	END_IF
	END_IF
	END_IF
END_IF

IF MovimentoVert_GA_0.StartWhat='Go_down' AND MovimentoVert_GA_0.State='Busy' THEN
	IF Richiesta_interna=TRUE OR Request_down= TRUE THEN
	IF P1Vis=TRUE THEN 
    IF 1>Destination AND Current>1 THEN
		Destination:=1;
		ELSIF 1<Destination AND Current_ok=TRUE THEN Destination:=1;
	END_IF
	END_IF
	END_IF
END_IF

IF MovimentoVert_GA_0.StartWhat='Go_down' AND MovimentoVert_GA_0.State='Busy' THEN
	IF Richiesta_interna=TRUE OR Request_down= TRUE THEN
	IF P2Vis=TRUE THEN 
    IF 2>Destination AND Current>2 THEN
		Destination:=2;
		ELSIF 2<Destination AND Current_ok=TRUE THEN Destination:=2;
	END_IF
	END_IF
	END_IF
END_IF

IF MovimentoVert_GA_0.StartWhat='Go_down' AND MovimentoVert_GA_0.State='Busy' THEN
	IF Richiesta_interna=TRUE OR Request_down= TRUE THEN
	IF P3Vis=TRUE THEN 
    IF 3>Destination AND Current>3 THEN
		Destination:=3;
		ELSIF 3<Destination AND Current_ok=TRUE THEN Destination:=3;
	END_IF
	END_IF
	END_IF
END_IF

IF MovimentoVert_GA_0.StartWhat='Go_down' AND MovimentoVert_GA_0.State='Busy' THEN
	IF Richiesta_interna=TRUE OR Request_down= TRUE THEN
	IF P4Vis=TRUE THEN 
    IF 4>Destination AND Current>4 THEN
		Destination:=4;
		ELSIF 4<Destination AND Current_ok=TRUE THEN Destination:=4;
	END_IF
	END_IF
	END_IF
END_IF

IF MovimentoVert_GA_0.StartWhat='Go_down' AND MovimentoVert_GA_0.State='Busy' THEN
	IF Richiesta_interna=TRUE OR Request_down= TRUE THEN
	IF P5Vis=TRUE THEN 
    IF 5>Destination AND Current>5 THEN
		Destination:=5;
		ELSIF 5<Destination AND Current_ok=TRUE THEN Destination:=5;
	END_IF
	END_IF
	END_IF
END_IF

IF MovimentoVert_GA_0.StartWhat='Go_down' AND MovimentoVert_GA_0.State='Busy' THEN
	IF Richiesta_interna=TRUE OR Request_down= TRUE THEN
	IF P6Vis=TRUE THEN 
    IF 6>Destination AND Current>6 THEN
		Destination:=6;
		ELSIF 6<Destination AND Current_ok=TRUE THEN Destination:=6;
	END_IF
	END_IF
	END_IF
END_IF

IF MovimentoVert_GA_0.StartWhat='Go_down' AND MovimentoVert_GA_0.State='Busy' THEN
	IF Richiesta_interna=TRUE OR Request_down= TRUE THEN
	IF P7Vis=TRUE THEN 
    IF 7>Destination AND Current>7 THEN
		Destination:=7;
		ELSIF 7<Destination AND Current_ok=TRUE THEN Destination:=7;
	END_IF
	END_IF
	END_IF
END_IF







//VIS ESTERNI UP

IF MovimentoVert_GA_0.StartWhat='Go_up' AND MovimentoVert_GA_0.State='Busy' THEN
	IF Richiesta_interna=TRUE OR Request_up= TRUE THEN
	IF UpDeckGVis=TRUE THEN 
    IF 0<Destination AND Current<0 THEN
		Destination:=0;
		ELSIF 0>Destination AND Current_ok=TRUE THEN Destination:=0;
	END_IF
	END_IF
	END_IF
END_IF

IF MovimentoVert_GA_0.StartWhat='Go_up' AND MovimentoVert_GA_0.State='Busy' THEN
	IF Richiesta_interna=TRUE OR Request_up= TRUE THEN
	IF UpDeck1Vis=TRUE THEN 
    IF 1<Destination AND Current<1 AND RS_counter<(2*(1-Piano_partenza)) THEN
		Destination:=1;
		ELSIF 1>Destination AND Current_ok=TRUE THEN Destination:=1;
	END_IF
	END_IF
	END_IF
END_IF

IF MovimentoVert_GA_0.StartWhat='Go_up' AND MovimentoVert_GA_0.State='Busy' THEN
	IF Richiesta_interna=TRUE OR Request_up= TRUE THEN
	IF UpDeck2Vis=TRUE THEN 
    IF 2<Destination AND Current<2 AND RS_counter<(2*(2-Piano_partenza)) THEN
		Destination:=2;
		ELSIF 2>Destination AND Current_ok=TRUE THEN Destination:=2;
	END_IF
	END_IF
	END_IF
END_IF

IF MovimentoVert_GA_0.StartWhat='Go_up' AND MovimentoVert_GA_0.State='Busy' THEN
	IF Richiesta_interna=TRUE OR Request_up= TRUE THEN
	IF UpDeck3Vis=TRUE THEN 
    IF 3<Destination AND Current<3 AND RS_counter<(2*(3-Piano_partenza)) THEN
		Destination:=3;
		ELSIF 3>Destination AND Current_ok=TRUE THEN Destination:=3;
	END_IF
	END_IF
	END_IF
END_IF

IF MovimentoVert_GA_0.StartWhat='Go_up' AND MovimentoVert_GA_0.State='Busy' THEN
	IF Richiesta_interna=TRUE OR Request_up= TRUE THEN
	IF UpDeck4Vis=TRUE THEN 
    IF 4<Destination AND Current<4 AND RS_counter<(2*(4-Piano_partenza)) THEN
		Destination:=4;
		ELSIF 4>Destination AND Current_ok=TRUE THEN Destination:=4;
	END_IF
	END_IF
	END_IF
END_IF

IF MovimentoVert_GA_0.StartWhat='Go_up' AND MovimentoVert_GA_0.State='Busy' THEN
	IF Richiesta_interna=TRUE OR Request_up= TRUE THEN
	IF UpDeck5Vis=TRUE THEN 
    IF 5<Destination AND Current<5 AND RS_counter<(2*(5-Piano_partenza)) THEN
		Destination:=5;
		ELSIF 5>Destination AND Current_ok=TRUE THEN Destination:=5;
	END_IF
	END_IF
	END_IF
END_IF

IF MovimentoVert_GA_0.StartWhat='Go_up' AND MovimentoVert_GA_0.State='Busy' THEN
	IF Richiesta_interna=TRUE OR Request_up= TRUE THEN
	IF UpDeck6Vis=TRUE THEN 
    IF 6<Destination AND Current<6 AND RS_counter<(2*(6-Piano_partenza)) THEN
		Destination:=6;
		ELSIF 6>Destination AND Current_ok=TRUE THEN Destination:=6;
	END_IF
	END_IF
	END_IF
END_IF

//VIS ESTERNI DOWN

IF MovimentoVert_GA_0.StartWhat='Go_down' AND MovimentoVert_GA_0.State='Busy' THEN
	IF Richiesta_interna=TRUE OR Request_down= TRUE THEN
	IF DownDeck1Vis=TRUE THEN 
    IF 1>Destination AND Current>1 AND RS_counter<(2*(Piano_partenza-1)) THEN
		Destination:=1;
		ELSIF 1<Destination AND Current_ok=TRUE THEN Destination:=1;
	END_IF
	END_IF
	END_IF
END_IF

IF MovimentoVert_GA_0.StartWhat='Go_down' AND MovimentoVert_GA_0.State='Busy' THEN
	IF Richiesta_interna=TRUE OR Request_down= TRUE THEN
	IF DownDeck2Vis=TRUE THEN 
    IF 2>Destination AND Current>2 AND RS_counter<(2*(Piano_partenza-2)) THEN
		Destination:=2;
		ELSIF 2<Destination AND Current_ok=TRUE THEN Destination:=2;
	END_IF
	END_IF
	END_IF
END_IF

IF MovimentoVert_GA_0.StartWhat='Go_down' AND MovimentoVert_GA_0.State='Busy' THEN
	IF Richiesta_interna=TRUE OR Request_down= TRUE THEN
	IF DownDeck3Vis=TRUE THEN 
    IF 3>Destination AND Current>3 AND RS_counter<(2*(Piano_partenza-3)) THEN
		Destination:=3;
		ELSIF 3<Destination AND Current_ok=TRUE THEN Destination:=3;
	END_IF
	END_IF
	END_IF
END_IF

IF MovimentoVert_GA_0.StartWhat='Go_down' AND MovimentoVert_GA_0.State='Busy' THEN
	IF Richiesta_interna=TRUE OR Request_down= TRUE THEN
	IF DownDeck4Vis=TRUE THEN 
    IF 4>Destination AND Current>4 AND RS_counter<(2*(Piano_partenza-4)) THEN
		Destination:=4;
		ELSIF 4<Destination AND Current_ok=TRUE THEN Destination:=4;
	END_IF
	END_IF
	END_IF
END_IF

IF MovimentoVert_GA_0.StartWhat='Go_down' AND MovimentoVert_GA_0.State='Busy' THEN
	IF Richiesta_interna=TRUE OR Request_down= TRUE THEN
	IF DownDeck5Vis=TRUE THEN 
    IF 5>Destination AND Current>5 AND RS_counter<(2*(Piano_partenza-5)) THEN
		Destination:=5;
		ELSIF 5<Destination AND Current_ok=TRUE THEN Destination:=5;
	END_IF
	END_IF
	END_IF
END_IF

IF MovimentoVert_GA_0.StartWhat='Go_down' AND MovimentoVert_GA_0.State='Busy' THEN
	IF Richiesta_interna=TRUE OR Request_down= TRUE THEN
	IF DownDeck6Vis=TRUE THEN 
    IF 6>Destination AND Current>6 AND RS_counter<(2*(Piano_partenza-6)) THEN
		Destination:=6;
		ELSIF 6<Destination AND Current_ok=TRUE THEN Destination:=6;
	END_IF
	END_IF
	END_IF
END_IF

IF MovimentoVert_GA_0.StartWhat='Go_down' AND MovimentoVert_GA_0.State='Busy' THEN
	IF Richiesta_interna=TRUE OR Request_down= TRUE THEN
	IF DownDeck7Vis=TRUE THEN 
    IF 7>Destination AND Current>7 THEN
		Destination:=7;
		ELSIF 7<Destination AND Current_ok=TRUE THEN Destination:=7;
	END_IF
	END_IF
	END_IF
END_IF


//MEMORIA CHIAMATE NON AL VOLO ESTERNO ALTO

IF MovimentoVert_GA_0.State='Ready' AND Chiamata_in_sospeso=TRUE THEN
	IF Richiesta_interna=TRUE OR Request_up= TRUE THEN
	IF UpDeckGVis=TRUE THEN 
    IF 0<Destination AND Current<0 THEN
		Destination:=0;
		ELSIF 0>Destination AND Current_ok=TRUE THEN Destination:=0;
	END_IF
	END_IF
	END_IF
END_IF

IF MovimentoVert_GA_0.State='Ready' AND Chiamata_in_sospeso=TRUE THEN
	IF Richiesta_interna=TRUE OR Request_up= TRUE THEN
	IF UpDeck1Vis=TRUE THEN 
    IF 1<Destination AND Current<1 THEN
		Destination:=1;
		ELSIF 1>Destination AND Current_ok=TRUE THEN Destination:=1;
	END_IF
	END_IF
	END_IF
END_IF

IF MovimentoVert_GA_0.State='Ready' AND Chiamata_in_sospeso=TRUE THEN
	IF Richiesta_interna=TRUE OR Request_up= TRUE THEN
	IF UpDeck2Vis=TRUE THEN 
    IF 2<Destination AND Current<2 THEN
		Destination:=2;
		ELSIF 2>Destination AND Current_ok=TRUE THEN Destination:=2;
	END_IF
	END_IF
	END_IF
END_IF

IF MovimentoVert_GA_0.State='Ready' AND Chiamata_in_sospeso=TRUE THEN
	IF Richiesta_interna=TRUE OR Request_up= TRUE THEN
	IF UpDeck3Vis=TRUE THEN 
    IF 3<Destination AND Current<3 THEN
		Destination:=3;
		ELSIF 3>Destination AND Current_ok=TRUE THEN Destination:=3;
	END_IF
	END_IF
	END_IF
END_IF

IF MovimentoVert_GA_0.State='Ready' AND Chiamata_in_sospeso=TRUE THEN
	IF Richiesta_interna=TRUE OR Request_up= TRUE THEN
	IF UpDeck4Vis=TRUE THEN 
    IF 4<Destination AND Current<4 THEN
		Destination:=4;
		ELSIF 4>Destination AND Current_ok=TRUE THEN Destination:=4;
	END_IF
	END_IF
	END_IF
END_IF

IF MovimentoVert_GA_0.State='Ready' AND Chiamata_in_sospeso=TRUE THEN
	IF Richiesta_interna=TRUE OR Request_up= TRUE THEN
	IF UpDeck5Vis=TRUE THEN 
    IF 5<Destination AND Current<5 THEN
		Destination:=5;
		ELSIF 5>Destination AND Current_ok=TRUE THEN Destination:=5;
	END_IF
	END_IF
	END_IF
END_IF

IF MovimentoVert_GA_0.State='Ready' AND Chiamata_in_sospeso=TRUE THEN
	IF Richiesta_interna=TRUE OR Request_up= TRUE THEN
	IF UpDeck6Vis=TRUE THEN 
    IF 6<Destination AND Current<6 THEN
		Destination:=6;
		ELSIF 6>Destination AND Current_ok=TRUE THEN Destination:=6;
	END_IF
	END_IF
	END_IF
END_IF

//MEMORIA CHIAMATE ESTERNO BASSO

IF MovimentoVert_GA_0.State='Ready' AND Chiamata_in_sospeso=TRUE THEN
	IF Richiesta_interna=TRUE OR Request_down= TRUE THEN
	IF DownDeck1Vis=TRUE THEN 
    IF 1>Destination AND Current>1 THEN
		Destination:=1;
		ELSIF 1<Destination AND Current_ok=TRUE THEN Destination:=1;
	END_IF
	END_IF
	END_IF
END_IF

IF MovimentoVert_GA_0.State='Ready' AND Chiamata_in_sospeso=TRUE THEN
	IF Richiesta_interna=TRUE OR Request_down= TRUE THEN
	IF DownDeck2Vis=TRUE THEN 
    IF 2>Destination AND Current>2 THEN
		Destination:=2;
		ELSIF 2<Destination AND Current_ok=TRUE THEN Destination:=2;
	END_IF
	END_IF
	END_IF
END_IF

IF MovimentoVert_GA_0.State='Ready' AND Chiamata_in_sospeso=TRUE THEN
	IF Richiesta_interna=TRUE OR Request_down= TRUE THEN
	IF DownDeck3Vis=TRUE THEN 
    IF 3>Destination AND Current>3 THEN
		Destination:=3;
		ELSIF 3<Destination AND Current_ok=TRUE THEN Destination:=3;
	END_IF
	END_IF
	END_IF
END_IF

IF MovimentoVert_GA_0.State='Ready' AND Chiamata_in_sospeso=TRUE THEN
	IF Richiesta_interna=TRUE OR Request_down= TRUE THEN
	IF DownDeck4Vis=TRUE THEN 
    IF 4>Destination AND Current>4 THEN
		Destination:=4;
		ELSIF 4<Destination AND Current_ok=TRUE THEN Destination:=4;
	END_IF
	END_IF
	END_IF
END_IF

IF MovimentoVert_GA_0.State='Ready' AND Chiamata_in_sospeso=TRUE THEN
	IF Richiesta_interna=TRUE OR Request_down= TRUE THEN
	IF DownDeck5Vis=TRUE THEN 
    IF 5>Destination AND Current>5 THEN
		Destination:=5;
		ELSIF 5<Destination AND Current_ok=TRUE THEN Destination:=5;
	END_IF
	END_IF
	END_IF
END_IF

IF MovimentoVert_GA_0.State='Ready' AND Chiamata_in_sospeso=TRUE THEN
	IF Richiesta_interna=TRUE OR Request_down= TRUE THEN
	IF DownDeck6Vis=TRUE THEN 
    IF 6>Destination AND Current>6 THEN
		Destination:=6;
		ELSIF 6<Destination AND Current_ok=TRUE THEN Destination:=6;
	END_IF
	END_IF
	END_IF
END_IF

IF MovimentoVert_GA_0.State='Ready' AND Chiamata_in_sospeso=TRUE THEN
	IF Richiesta_interna=TRUE OR Request_down= TRUE THEN
	IF DownDeck7Vis=TRUE THEN 
    IF 7>Destination AND Current>7 THEN
		Destination:=7;
		ELSIF 7<Destination AND Current_ok=TRUE THEN Destination:=7;
	END_IF
	END_IF
	END_IF
END_IF

//MEMORIA CHIAMATE INTERNE ALTO

IF MovimentoVert_GA_0.State='Ready' AND Chiamata_in_sospeso=TRUE THEN
	IF Richiesta_interna=TRUE OR Request_up= TRUE THEN
	IF PGVis=TRUE THEN 
    IF 0<Destination AND Current<0 THEN
		Destination:=0;
		ELSIF 0>Destination AND Current_ok=TRUE THEN Destination:=0;
	END_IF
	END_IF
	END_IF
END_IF

IF MovimentoVert_GA_0.State='Ready' AND Chiamata_in_sospeso=TRUE THEN
	IF Richiesta_interna=TRUE OR Request_up= TRUE THEN
	IF P1Vis=TRUE THEN 
    IF 1<Destination AND Current<1 THEN
		Destination:=1;
		ELSIF 1>Destination AND Current_ok=TRUE THEN Destination:=1;
	END_IF
	END_IF
	END_IF
END_IF

IF MovimentoVert_GA_0.State='Ready' AND Chiamata_in_sospeso=TRUE THEN
	IF Richiesta_interna=TRUE OR Request_up= TRUE THEN
	IF P2Vis=TRUE THEN 
    IF 2<Destination AND Current<2 THEN
		Destination:=2;
		ELSIF 2>Destination AND Current_ok=TRUE THEN Destination:=2;
	END_IF
	END_IF
	END_IF
END_IF

IF MovimentoVert_GA_0.State='Ready' AND Chiamata_in_sospeso=TRUE THEN
	IF Richiesta_interna=TRUE OR Request_up= TRUE THEN
	IF P3Vis=TRUE THEN 
    IF 3<Destination AND Current<3 THEN
		Destination:=3;
		ELSIF 3>Destination AND Current_ok=TRUE THEN Destination:=3;
	END_IF
	END_IF
	END_IF
END_IF

IF MovimentoVert_GA_0.State='Ready' AND Chiamata_in_sospeso=TRUE THEN
	IF Richiesta_interna=TRUE OR Request_up= TRUE THEN
	IF P4Vis=TRUE THEN 
    IF 4<Destination AND Current<4 THEN
		Destination:=4;
		ELSIF 4>Destination AND Current_ok=TRUE THEN Destination:=4;
	END_IF
	END_IF
	END_IF
END_IF

IF MovimentoVert_GA_0.State='Ready' AND Chiamata_in_sospeso=TRUE THEN
	IF Richiesta_interna=TRUE OR Request_up= TRUE THEN
	IF P5Vis=TRUE THEN 
    IF 5<Destination AND Current<5 THEN
		Destination:=5;
		ELSIF 5>Destination AND Current_ok=TRUE THEN Destination:=5;
	END_IF
	END_IF
	END_IF
END_IF

IF MovimentoVert_GA_0.State='Ready' AND Chiamata_in_sospeso=TRUE THEN
	IF Richiesta_interna=TRUE OR Request_up= TRUE THEN
	IF P6Vis=TRUE THEN 
    IF 6<Destination AND Current<6 THEN
		Destination:=6;
		ELSIF 6>Destination AND Current_ok=TRUE THEN Destination:=6;
	END_IF
	END_IF
	END_IF
END_IF

IF MovimentoVert_GA_0.State='Ready' AND Chiamata_in_sospeso=TRUE THEN
	IF Richiesta_interna=TRUE OR Request_up= TRUE THEN
	IF P7Vis=TRUE THEN 
    IF 7<Destination AND Current<7 THEN
		Destination:=7;
		ELSIF 7>Destination AND Current_ok=TRUE THEN Destination:=7;
	END_IF
	END_IF
	END_IF
END_IF

//MEMORIA CHIAMATE INTERNE BASSO

IF MovimentoVert_GA_0.State='Ready' AND Chiamata_in_sospeso=TRUE THEN
	IF Richiesta_interna=TRUE OR Request_down= TRUE THEN
	IF PGVis=TRUE THEN 
    IF 0>Destination AND Current>0 THEN
		Destination:=0;
		ELSIF 0<Destination AND Current_ok=TRUE THEN Destination:=0;
	END_IF
	END_IF
	END_IF
END_IF

IF MovimentoVert_GA_0.State='Ready' AND Chiamata_in_sospeso=TRUE THEN
	IF Richiesta_interna=TRUE OR Request_down= TRUE THEN
	IF P1Vis=TRUE THEN 
    IF 1>Destination AND Current>1 THEN
		Destination:=1;
		ELSIF 1<Destination AND Current_ok=TRUE THEN Destination:=1;
	END_IF
	END_IF
	END_IF
END_IF

IF MovimentoVert_GA_0.State='Ready' AND Chiamata_in_sospeso=TRUE THEN
	IF Richiesta_interna=TRUE OR Request_down= TRUE THEN
	IF P2Vis=TRUE THEN 
    IF 2>Destination AND Current>2 THEN
		Destination:=2;
		ELSIF 2<Destination AND Current_ok=TRUE THEN Destination:=2;
	END_IF
	END_IF
	END_IF
END_IF

IF MovimentoVert_GA_0.State='Ready' AND Chiamata_in_sospeso=TRUE THEN
	IF Richiesta_interna=TRUE OR Request_down= TRUE THEN
	IF P3Vis=TRUE THEN 
    IF 3>Destination AND Current>3 THEN
		Destination:=3;
		ELSIF 3<Destination AND Current_ok=TRUE THEN Destination:=3;
	END_IF
	END_IF
	END_IF
END_IF

IF MovimentoVert_GA_0.State='Ready' AND Chiamata_in_sospeso=TRUE THEN
	IF Richiesta_interna=TRUE OR Request_down= TRUE THEN
	IF P4Vis=TRUE THEN 
    IF 4>Destination AND Current>4 THEN
		Destination:=4;
		ELSIF 4<Destination AND Current_ok=TRUE THEN Destination:=4;
	END_IF
	END_IF
	END_IF
END_IF

IF MovimentoVert_GA_0.State='Ready' AND Chiamata_in_sospeso=TRUE THEN
	IF Richiesta_interna=TRUE OR Request_down= TRUE THEN
	IF P5Vis=TRUE THEN 
    IF 5>Destination AND Current>5 THEN
		Destination:=5;
		ELSIF 5<Destination AND Current_ok=TRUE THEN Destination:=5;
	END_IF
	END_IF
	END_IF
END_IF

IF MovimentoVert_GA_0.State='Ready' AND Chiamata_in_sospeso=TRUE THEN
	IF Richiesta_interna=TRUE OR Request_down= TRUE THEN
	IF P6Vis=TRUE THEN 
    IF 6>Destination AND Current>6 THEN
		Destination:=6;
		ELSIF 6<Destination AND Current_ok=TRUE THEN Destination:=6;
	END_IF
	END_IF
	END_IF
END_IF

IF MovimentoVert_GA_0.State='Ready' AND Chiamata_in_sospeso=TRUE THEN
	IF Richiesta_interna=TRUE OR Request_down= TRUE THEN
	IF P7Vis=TRUE THEN 
    IF 7>Destination AND Current>7 THEN
		Destination:=7;
		ELSIF 7<Destination AND Current_ok=TRUE THEN Destination:=7;
	END_IF
	END_IF
	END_IF
END_IF


//REGOLE FINALI


IF Request_down=FALSE AND MovimentoVert_GA_0.State='Ready' AND Chiamata_in_sospeso=TRUE THEN
	IF Request_up=TRUE AND Richiesta_interna=FALSE THEN
	IF UpDeckGVis=TRUE THEN Destination:=0;
    ELSIF UpDeck1Vis=TRUE THEN Destination:=1;
	ELSIF UpDeck2Vis=TRUE THEN Destination:=2;
	ELSIF UpDeck3Vis=TRUE THEN Destination:=3;
	ELSIF UpDeck4Vis=TRUE THEN Destination:=4;
	ELSIF UpDeck5Vis=TRUE THEN Destination:=5;
	ELSIF UpDeck6Vis=TRUE THEN Destination:=6;
	END_IF
	END_IF
END_IF

IF Request_up=FALSE AND MovimentoVert_GA_0.State='Ready' AND Chiamata_in_sospeso=TRUE THEN
	IF Request_down=TRUE AND Richiesta_interna=FALSE THEN
	IF DownDeck7Vis=TRUE THEN Destination:=7;
	ELSIF DownDeck6Vis=TRUE THEN Destination:=6;
	ELSIF DownDeck5Vis=TRUE THEN Destination:=5;
	ELSIF DownDeck4Vis=TRUE THEN Destination:=4;
	ELSIF DownDeck3Vis=TRUE THEN Destination:=3;
	ELSIF DownDeck2Vis=TRUE THEN Destination:=2;
	ELSIF DownDeck1Vis=TRUE THEN Destination:=1;
	END_IF
	END_IF
END_IF

IF Request_up=TRUE AND Request_down=TRUE AND Richiesta_interna=FALSE AND MovimentoVert_GA_0.State='Ready' THEN
	IF UpDeckGVis=TRUE THEN Destination:=0;
    ELSIF UpDeck1Vis=TRUE THEN Destination:=1;
	ELSIF UpDeck2Vis=TRUE THEN Destination:=2;
	ELSIF UpDeck3Vis=TRUE THEN Destination:=3;
	ELSIF UpDeck4Vis=TRUE THEN Destination:=4;
	ELSIF UpDeck5Vis=TRUE THEN Destination:=5;
	ELSIF UpDeck6Vis=TRUE THEN Destination:=6;
	END_IF
END_IF
END_ACTION

ACTION _aMoto_verticale_active_1:
//REGOLAZIONE VELOCITA'
IF RS_counter=0 AND Current=-1 THEN
	Piano_partenza:=Current+1;
END_IF

IF RS_counter=0 AND Current>-1 THEN
	Piano_partenza:=Current;
END_IF

IF RampSensor=TRUE AND t_ramp=0 THEN
	RS_counter:=RS_counter+1;
	Ramp_counter:=Ramp_counter+1; //Variabile per il guasto dei magnetini(affrontata in dettaglio in memoria chiamate
END_IF

IF RampSensor=TRUE THEN
	t_ramp:=t_ramp+1;
END_IF

IF RampSensor=FALSE THEN
	t_ramp:=0;
END_IF

IF RampSensor=FALSE AND RS_counter=0 THEN
	VEL:=FALSE;
END_IF

IF RS_counter=1 THEN
	VEL:=TRUE;
END_IF

IF Destination=0 THEN
    IF RS_counter=2*Piano_partenza THEN
		VEL:=FALSE;
    END_IF
END_IF

IF Destination>0 AND Piano_partenza=0 THEN
	IF RS_counter=2*Destination THEN
		VEL:=FALSE;
    END_IF
END_IF

IF Destination>0 AND Piano_partenza>0 AND Piano_partenza>Destination THEN
	IF RS_counter=(Piano_partenza-Destination)*2 THEN
		VEL:=FALSE;
	END_IF
END_IF

IF Destination>0 AND Piano_partenza>0 AND Piano_partenza<Destination THEN
	IF RS_counter=(Destination-Piano_partenza)*2 THEN
		VEL:=FALSE;
	END_IF
END_IF

//ACCENSIONE E SPEGNIMENTO MOTO
IF Current<Destination AND MovimentoVert_GA_0.State='Ready' THEN
	MovimentoVert_GA_0.Start:=TRUE;
	MovimentoVert_GA_0.Stop:=FALSE;
	MovimentoVert_GA_0.StartWhat:='Go_up';
END_IF
IF Current>Destination AND MovimentoVert_GA_0.State='Ready' THEN
	MovimentoVert_GA_0.Start:=TRUE;
	MovimentoVert_GA_0.Stop:=FALSE;
	MovimentoVert_GA_0.StartWhat:='Go_down';
END_IF

IF DeckSensor=TRUE AND MovimentoVert_GA_0.State='Busy' THEN  
	IF Current>Destination AND t_deck=0 THEN
		Current:=Current-1;
		Deck_counter:=Deck_counter+1; //Variabile per il guasto dei magnetini
	ELSIF Current<Destination AND t_deck=0 THEN
		Current:=Current+1;
		Deck_counter:=Deck_counter+1;
	END_IF
		t_deck:=t_deck+1;  //Variabile per contare una sola volta il decksensor
END_IF


IF DeckSensor=FALSE THEN
	t_deck:=0;
END_IF


IF (Current=Destination) THEN
	MovimentoVert_GA_0.Stop:= TRUE;
	MovimentoVert_GA_0.Start:= FALSE;
    Current_Ok:=TRUE;
	Deck_counter:=0;
	Ramp_counter:=0;
END_IF
END_ACTION

ACTION _aChiusura_P_exit:
OpFatta := FALSE;
END_ACTION

ACTION _aChiusura_P_active:
IF Doors_GA_0.State='ready' THEN
	Doors_GA_0.Do_:=TRUE;
	Doors_GA_0.DoWhat:='Chiusura';
END_IF

IF (Doors_GA_0.Done= TRUE) AND Doors_GA_0.State='Busy' THEN
	Doors_GA_0.Do_:=FALSE;
	OpFatta:=TRUE;
END_IF
END_ACTION

ACTION _aMoto_verticale_entry:
Current_ok:= FALSE;
END_ACTION

END_PROGRAM

// Device/Application/Visualization
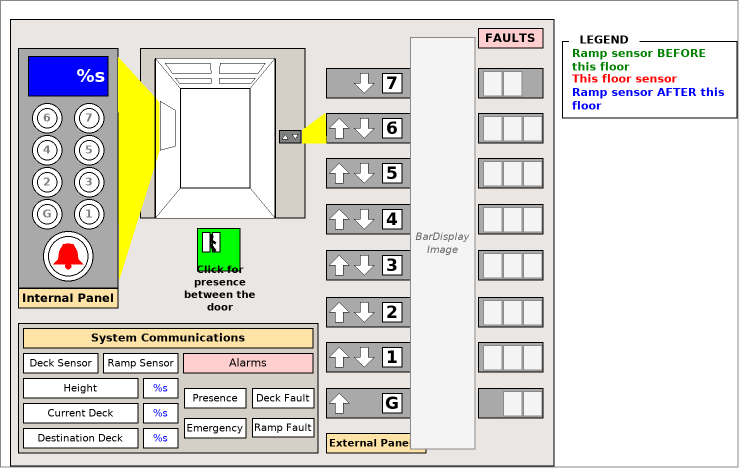
VISUALIZATION Visualization  // 739x468
    Rectangle (10,19 544x447)
    Rectangle (197,228 43x43), colour toggle: GVL.Presence
    Rectangle (18,323 300x130)
    Rectangle (326,433 100x20), "External Panels"
    Rectangle (326,342 100x30)
    Rectangle (382,347 20x20), "1"
    Polygon (354,357) (360,357) (360,347) (368,347) (368,357) (374,357) (364,367), colour toggle: GVL.DownDeck1Vis
        tap GVL.DownDeck1
    Polygon (329,357) (335,357) (335,367) (343,367) (343,357) (349,357) (339,347), colour toggle: GVL.UpDeck1Vis
        tap GVL.UpDeck1
    Rectangle (326,297 100x30)
    Rectangle (382,302 20x20), "2"
    Polygon (354,312) (360,312) (360,302) (368,302) (368,312) (374,312) (364,322), colour toggle: GVL.DownDeck2Vis
        tap GVL.DownDeck2
    Polygon (329,312) (335,312) (335,322) (343,322) (343,312) (349,312) (339,302), colour toggle: GVL.UpDeck2Vis
        tap GVL.UpDeck2
    Rectangle (326,250 100x30)
    Rectangle (382,255 20x20), "3"
    Polygon (354,265) (360,265) (360,255) (368,255) (368,265) (374,265) (364,275), colour toggle: GVL.DownDeck3Vis
        tap GVL.DownDeck3
    Polygon (329,265) (335,265) (335,275) (343,275) (343,265) (349,265) (339,255), colour toggle: GVL.UpDeck3Vis
        tap GVL.UpDeck3
    Rectangle (326,204 100x30)
    Rectangle (382,209 20x20), "4"
    Polygon (354,219) (360,219) (360,209) (368,209) (368,219) (374,219) (364,229), colour toggle: GVL.DownDeck4Vis
        tap GVL.DownDeck4
    Polygon (329,219) (335,219) (335,229) (343,229) (343,219) (349,219) (339,209), colour toggle: GVL.UpDeck4Vis
        tap GVL.UpDeck4
    Rectangle (326,158 100x30)
    Rectangle (382,163 20x20), "5"
    Polygon (354,173) (360,173) (360,163) (368,163) (368,173) (374,173) (364,183), colour toggle: GVL.DownDeck5Vis
        tap GVL.DownDeck5
    Polygon (329,173) (335,173) (335,183) (343,183) (343,173) (349,173) (339,163), colour toggle: GVL.UpDeck5Vis
        tap GVL.UpDeck5
    Rectangle (326,113 100x30)
    Rectangle (382,118 20x20), "6"
    Polygon (354,128) (360,128) (360,118) (368,118) (368,128) (374,128) (364,138), colour toggle: GVL.DownDeck6Vis
        tap GVL.DownDeck6
    Polygon (329,128) (335,128) (335,138) (343,138) (343,128) (349,128) (339,118), colour toggle: GVL.UpDeck6Vis
        tap GVL.UpDeck6
    Rectangle (326,68 100x30)
    Rectangle (382,73 20x20), "7"
    Polygon (354,83) (360,83) (360,73) (368,73) (368,83) (374,83) (364,93), colour toggle: GVL.DownDeck7Vis
        tap GVL.DownDeck7
    Rectangle (326,388 100x30)
    Rectangle (382,393 20x20), "G"
    Polygon (329,403) (335,403) (335,413) (343,413) (343,403) (349,403) (339,393), colour toggle: GVL.UpDeckGVis
        tap GVL.UpDeckG
    RoundedRectangle (18,48 100x240)
    Rectangle (18,288 100x20), "Internal Panel"
    Ellipse (74,199 30x30), colour toggle: GVL.P1Vis
    Ellipse (79,204 20x20), "1"
        tap GVL.P1
    Ellipse (32,199 30x30), colour toggle: GVL.PGVis
    Ellipse (37,204 20x20), "G"
        tap GVL.PG
    Ellipse (74,167 30x30), colour toggle: GVL.P3Vis
    Ellipse (79,172 20x20), "3"
        tap GVL.P3
    Ellipse (32,167 30x30), colour toggle: GVL.P2Vis
    Ellipse (37,172 20x20), "2"
        tap GVL.P2
    Ellipse (74,135 30x30), colour toggle: GVL.P5Vis
    Ellipse (79,140 20x20), "5"
        tap GVL.P5
    Ellipse (32,135 30x30), colour toggle: GVL.P4Vis
    Ellipse (37,140 20x20), "4"
        tap GVL.P4
    Ellipse (74,103 30x30), colour toggle: GVL.P7Vis
    Ellipse (79,108 20x20), "7"
        tap GVL.P7
    Ellipse (32,103 30x30), colour toggle: GVL.P6Vis
    Ellipse (37,108 20x20), "6"
        tap GVL.P6
    Rectangle (28,56 80x40), "%s", text variable: GVL.Destination
    Ellipse (43,231 50x50), tooltip "EMERGENCY", colour toggle: GVL.Emergency
    Group (48,236 40x40)
        toggle GVL.Emergency
        Ellipse (0,0 40x40), tooltip "EMERGENCY"
        Polygon (5,28) (10,23) (11,15) (15,8) (20,7) (25,8) (29,15) (30,23) (35,28)
        Ellipse (17,27 6x6)
    Polygon (35,72) (45,62) (55,72), colour toggle: GVL.Motor_on AND GVL.Up
    Polygon (35,80) (45,90) (55,80), colour toggle: GVL.Motor_on AND NOT GVL.Up
    Group (140,48 165x170)
        Rectangle (0,0 165x170)
        Rectangle (15,10 120x160)
        Polygon (40,40) (15,10) (135,10) (110,40)
        Rectangle (40,40 70x100)
        Polygon (15,170) (40,140) (110,140) (135,170)
        Polygon (20,102) (20,53) (35,62) (35,98)
        Polygon (79,35) (79,30) (115,30) (111,35)
        Polygon (39,35) (35,30) (71,30) (71,35)
        Polygon (32,25) (25,15) (70,15) (71,25)
        Polygon (79,25) (80,15) (125,15) (118,25)
        Group (139,82 22x13)
            Rectangle (0,0 22x13)
            Polygon (3,9) (6,4) (9,9)
            Polygon (13,4) (16,9) (19,4)
    BarDisplayImage (410,37 65x412), value: GVL.Height, style: BarDisplayImage-Gray, scale format: %.0f, scale -20..160
        p3451962224: VisuNativeControl.IP_Offline.Browser
    Rectangle (478,68 65x30)
    Rectangle (478,342 65x30)
    Rectangle (478,297 65x30)
    Rectangle (478,250 65x30)
    Rectangle (478,204 65x30)
    Rectangle (478,158 65x30)
    Rectangle (478,113 65x30)
    Rectangle (478,388 65x30)
    RockerSwitch (483,345 19x25), variable: GVL.Ramp1Down, behaviour: TOGGLE, style: Switch-RockerSwitch-Green
    RockerSwitch (503,345 19x25), variable: GVL.Sensor1, behaviour: TOGGLE, style: Switch-RockerSwitch-Red
    RockerSwitch (523,345 19x25), variable: GVL.Ramp1Up, behaviour: TOGGLE, style: Switch-RockerSwitch-Blue
    RockerSwitch (483,300 19x25), variable: GVL.Ramp2Down, behaviour: TOGGLE, style: Switch-RockerSwitch-Green
    RockerSwitch (503,300 19x25), variable: GVL.Sensor2, behaviour: TOGGLE, style: Switch-RockerSwitch-Red
    RockerSwitch (523,300 19x25), variable: GVL.Ramp2Up, behaviour: TOGGLE, style: Switch-RockerSwitch-Blue
    RockerSwitch (483,253 19x25), variable: GVL.Ramp3Down, behaviour: TOGGLE, style: Switch-RockerSwitch-Green
    RockerSwitch (503,253 19x25), variable: GVL.Sensor3, behaviour: TOGGLE, style: Switch-RockerSwitch-Red
    RockerSwitch (523,253 19x25), variable: GVL.Ramp3Up, behaviour: TOGGLE, style: Switch-RockerSwitch-Blue
    RockerSwitch (483,207 19x25), variable: GVL.Ramp4Down, behaviour: TOGGLE, style: Switch-RockerSwitch-Green
    RockerSwitch (503,207 19x25), variable: GVL.Sensor4, behaviour: TOGGLE, style: Switch-RockerSwitch-Red
    RockerSwitch (523,207 19x25), variable: GVL.Ramp4Up, behaviour: TOGGLE, style: Switch-RockerSwitch-Blue
    RockerSwitch (483,161 19x25), variable: GVL.Ramp5Down, behaviour: TOGGLE, style: Switch-RockerSwitch-Green
    RockerSwitch (503,161 19x25), variable: GVL.Sensor5, behaviour: TOGGLE, style: Switch-RockerSwitch-Red
    RockerSwitch (523,161 19x25), variable: GVL.Ramp5Up, behaviour: TOGGLE, style: Switch-RockerSwitch-Blue
    RockerSwitch (483,116 19x25), variable: GVL.Ramp6Down, behaviour: TOGGLE, style: Switch-RockerSwitch-Green
    RockerSwitch (503,116 19x25), variable: GVL.Sensor6, behaviour: TOGGLE, style: Switch-RockerSwitch-Red
    RockerSwitch (523,116 19x25), variable: GVL.Ramp6Up, behaviour: TOGGLE, style: Switch-RockerSwitch-Blue
    RockerSwitch (483,71 19x25), variable: GVL.Ramp7Down, behaviour: TOGGLE, style: Switch-RockerSwitch-Green
    RockerSwitch (503,71 19x25), variable: GVL.Sensor7, behaviour: TOGGLE, style: Switch-RockerSwitch-Red
    RockerSwitch (503,391 19x25), variable: GVL.SensorG, behaviour: TOGGLE, style: Switch-RockerSwitch-Red
    RockerSwitch (523,391 19x25), variable: GVL.RampGUp, behaviour: TOGGLE, style: Switch-RockerSwitch-Blue
    Rectangle (478,28 65x20), "FAULTS"
    Polygon (302,130) (325,113) (326,143) (302,143), invisible if: (GVL.Closing OR GVL.Opening) OR GVL.Closed
    Polygon (118,57) (159,102) (159,151) (119,279), invisible if: (GVL.Closing OR GVL.Opening) OR GVL.Closed
    Rectangle (155,58 0x160)
        p3528305787: GVL.Door
    Rectangle (275,58 0x160)
        p3528305787: -GVL.Door
    Rectangle (23,328 290x20), "System Communications"
    Rectangle (183,353 130x20), "Alarms"
    Rectangle (23,353 75x20), "Deck Sensor", colour toggle: GVL.DeckSensor
    Rectangle (143,378 35x20), "%s", text variable: GVL.Height
    Rectangle (184,388 62x20), "Presence", colour toggle: GVL.Presence
    Rectangle (103,353 75x20), "Ramp Sensor", colour toggle: GVL.RampSensor
    Rectangle (143,403 35x20), "%s", text variable: GVL.Current
    Rectangle (143,428 35x20), "%s", text variable: GVL.Destination
    Rectangle (252,388 62x20), "Deck Fault", colour toggle: GVL.FaultSensorAlarm
    Rectangle (184,418 62x20), "Emergency", colour toggle: GVL.EmergencyVis
    Rectangle (252,418 62x19), "Ramp Fault", colour toggle: GVL.FaultRampAlarm
    Rectangle (23,378 115x20), "Height"
    Rectangle (23,403 115x20), "Current Deck"
    Rectangle (23,428 115x20), "Destination Deck"
    Group (562,25 175x93)
        Rectangle (0,16 175x77)
        Rectangle (7,39 160x30), "This floor sensor"
        Rectangle (7,59 160x30), "Ramp sensor AFTER this floor"
        Rectangle (7,0 70x30), "LEGEND"
        Rectangle (7,20 160x30), "Ramp sensor BEFORE this floor"
    Group (202,232 33x34)
        toggle GVL.Presence
        Rectangle (10,0 8x20)
        Polygon (5,10) (12,20) (14,18) (5,6)
        Ellipse (6,2 5x5)
        Polygon (4,8) (13,12) (14,10) (4,4)
        Rectangle (0,0 8x20)
    Rectangle (169,273 102x31), "Click for presence between the door"
END_VISUALIZATION
